// TIA Portal V19 export
TYPE "LEXCHANGETRAY_typeAxisSimpleControlTorqueLimit"
// stored: Access Published
   STRUCT
      limit : LReal;
      mode : DInt;   // 0:力矩限制 1:固定挡块检测
   END_STRUCT;
END_TYPE
